{attribute addProperty BoxType "KL6551"}
{attribute addProperty Id "Parameter_StatusAT %I*UINT000Input_Data_1AT %I*USINT000Input_Data_2AT %I*USINT000Input_Data_3AT %I*USINT000Input_Data_4AT %I*USINT000Input_Data_5AT %I*USINT000Input_Data_6AT %I*USINT000Input_Data_7AT %I*USINT000Input_Data_8AT %I*USINT000Input_Data_9AT %I*USINT000Input_Data_10AT %I*USINT000Parameter_ControlAT %Q*UINT000Output_Data_1AT %Q*USINT000Output_Data_2AT %Q*USINT000Output_Data_3AT %Q*USINT000Output_Data_4AT %Q*USINT000Output_Data_5AT %Q*USINT000Output_Data_6AT %Q*USINT000Output_Data_7AT %Q*USINT000Output_Data_8AT %Q*USINT000Output_Data_9AT %Q*USINT000Output_Data_10AT %Q*USINT000"}
{attribute addProperty CRC "3607986224"}
{attribute addProperty SizeInBites "0"}
{attribute addProperty SizeInBytes "0"}
TYPE Channel_D70D8030 :
STRUCT
	{attribute addProperty Name "Parameter_Status"}
	Parameter_Status AT %I* : UINT;
	{attribute addProperty Name "Input_Data_1"}
	Input_Data_1 AT %I* : USINT;
	{attribute addProperty Name "Input_Data_2"}
	Input_Data_2 AT %I* : USINT;
	{attribute addProperty Name "Input_Data_3"}
	Input_Data_3 AT %I* : USINT;
	{attribute addProperty Name "Input_Data_4"}
	Input_Data_4 AT %I* : USINT;
	{attribute addProperty Name "Input_Data_5"}
	Input_Data_5 AT %I* : USINT;
	{attribute addProperty Name "Input_Data_6"}
	Input_Data_6 AT %I* : USINT;
	{attribute addProperty Name "Input_Data_7"}
	Input_Data_7 AT %I* : USINT;
	{attribute addProperty Name "Input_Data_8"}
	Input_Data_8 AT %I* : USINT;
	{attribute addProperty Name "Input_Data_9"}
	Input_Data_9 AT %I* : USINT;
	{attribute addProperty Name "Input_Data_10"}
	Input_Data_10 AT %I* : USINT;
	{attribute addProperty Name "Parameter_Control"}
	Parameter_Control AT %Q* : UINT;
	{attribute addProperty Name "Output_Data_1"}
	Output_Data_1 AT %Q* : USINT;
	{attribute addProperty Name "Output_Data_2"}
	Output_Data_2 AT %Q* : USINT;
	{attribute addProperty Name "Output_Data_3"}
	Output_Data_3 AT %Q* : USINT;
	{attribute addProperty Name "Output_Data_4"}
	Output_Data_4 AT %Q* : USINT;
	{attribute addProperty Name "Output_Data_5"}
	Output_Data_5 AT %Q* : USINT;
	{attribute addProperty Name "Output_Data_6"}
	Output_Data_6 AT %Q* : USINT;
	{attribute addProperty Name "Output_Data_7"}
	Output_Data_7 AT %Q* : USINT;
	{attribute addProperty Name "Output_Data_8"}
	Output_Data_8 AT %Q* : USINT;
	{attribute addProperty Name "Output_Data_9"}
	Output_Data_9 AT %Q* : USINT;
	{attribute addProperty Name "Output_Data_10"}
	Output_Data_10 AT %Q* : USINT;
END_STRUCT
END_TYPE

(* stored: Version 1.2.0.0, ProductVersion 3.1.4024.9
   DUT Channel_D70D8030: Id {de7bf141-224a-427b-bb19-222d177453fa} *)
